// Settings for GreenMaster
TYPE GreenMasterSettings :
STRUCT
RemoteStart :  WORD := 1; //  Remote (WebPort) unit activation (0=unit off, 1=normal speed, 2=high speed)
ResetAlarms :  BOOL :=FALSE; //  Reset alarms
Temperature_SP :  LREAL :=20.0; //  Temperature Set Point, C
TemperatureControlPV :  INT :=0; //  0 = Use T.BT1, 1 = Use F.BT1
SetPointOffsetCurve :  SetPointOffsetCurve; // Outdoorcompensation temperature


















TemperatureControl_P :  REAL :=0.05; //  Temperature control P
TemperatureControl_I :  TIME :=T#2M; //  Temperature control I
TemperatureControl_D :  TIME :=T#0M; //  Temperature control D
StartupHeatRecoveryTime :  TIME :=T#0M; //  Time at startup to recover
PostFireVentilationTime :  TIME :=T#1M; //  Time to ventilate when returning to operation after fire alarm
SupplyFanControlMode :  FanControlTypes ; //  Control mode (0=Pressure/T.BP1, 1=Flow/T.BF1) for Supply Air
SupplyFan_SP :  REAL :=100 ; //  Supply air control Set Point
SupplyFanHighSpeed_SP :  REAL ; //  Supply air control high speed Set Point
SupplyFanControl_P :  REAL :=0.002; //  Supply air control P
SupplyFanControl_I :  TIME :=T#2M; //  Supply air control I
ExtractFanControlMode :  FanControlTypes ; //  Control mode (0=Pressure/F.BP1, 1=Flow/F.BF1) for Extract Air
ExtractFan_SP :  REAL := 100; //  Extract air control Set Point
ExtractFanHighSpeed_SP :  REAL ; //  Extract air control high speed Set Point
ExtractFanControl_P :  REAL :=0.002; //  Extract air control P
ExtractFanControl_I :  TIME :=T#2M; //  Extract air control I
NightCoolingEN :  BOOL :=FALSE; //  Use Night cooling
NightCoolingTemperatureSP :  REAL :=18.0; //  Night cooling temperature Set Point, C
FanStopDelayTime :  TIME :=T#2M; //  Fan stop delay cool down period
WatchdogEnabled :  BOOL :=FALSE; //  Watchdog enable - enables unit on watchdog update failure 
Watchdog :  INT :=0; //  Watchdog counter to be changed at a minimum every 5 minutes (when enabled)  
NightCooling_V :  BOOL; //  Activate nigh time cooling  
TX1_M :  BOOL; // Heat exchanger manual override
T_GQ1_M :  BOOL; //  Supply air fan control manual override
F_GQ1_M :  BOOL; //  Extract air fan control manual override
C_QN1_M :  BOOL; //  Cool supply control valve manual override
H_QN1_M :  BOOL; //  Heat supply control valve manual override
TX1_OPM :  REAL; //  Heat exchanger manual value
T_GQ1_OPM :  REAL; //  Supply air fan control manual value
F_GQ1_OPM :  REAL; //  Extract air fan control manual value
C_QN1_OPM :  REAL; //  Cool supply control valve manual value
H_QN1_OPM :  REAL; //  Heat supply control valve manual value
END_STRUCT
END_TYPE

(* stored: Version 1.1.0.1, ProductVersion 3.1.4024.6
   DUT GreenMasterSettings: Id {3a990bac-3338-4d86-af98-b9811c6ccb8c} *)
